Staubli VAL3: BinToDec.pgx

public program BinToDec(string x_sBinary, num& x_nDecimal[])
  local num l_nNumBit
begin
  //-----------------------------------------------------------------------
  //Header begin
  //Description of program
  //  This program turns a binary word into a Decimal number
  //  Receives the binary word, verifies that the value is a
  //  binary value and turns it into the corresponding decimal
  //  number.
  //
  //Input parameters
  //  string x_sBinary :
  //    role : Binary value to convert
  //
  //Output parameters
  //  num x_nDecimal :
  //    role : Decimal value converted
  //
  //Example
  //  BinToDec("101110",nDecimalValue)
  //
  //History
  //  Creation : 16-04-09 - t.Gra
  //Header end
  //-----------------------------------------------------------------------
  //Initialization
  bRead=true
  l_nNumBit=0
  //chek the binary number is true and transforms this
  for l_nNumBit=(len(x_sBinary)-1) to 0 step -1
    if mid(x_sBinary,1,l_nNumBit)=="1"
      x_nDecimal=x_nDecimal+exp(((len(x_sBinary)-1)-l_nNumBit)*ln(2))
    elseIf mid(x_sBinary,1,l_nNumBit)=="0"
    else
      bRead=false
      x_nDecimal=0
    endIf
  endFor
end
